FUNCTION_BLOCK FB_ComputeFromImage
VAR_INPUT
	ptrXValues	: POINTER TO ARRAY[1..GVL.NumberVisionPoints] OF REAL;
	ptrYValues	: POINTER TO ARRAY[1..GVL.NumberVisionPoints] OF REAL;
	minor		: LREAL;	// in mm
	pitch		: LREAL;	// mm per pixel
END_VAR
VAR_OUTPUT
	centerX		: LREAL;
	centerY		: LREAL;
	a			: LREAL;	// major in mm
	b			: LREAL;	// minor in mm
END_VAR
	
VAR
	fbSecond	: FB_SecondOrder;
	fbFourth	: FB_FourthOrder;
	fbEllipse	: FB_Ellipse;
	xPeak		: LREAL;
	yPeak		: LREAL;
	XMirror		: ARRAY[1..GVL.NumberEllipsePoints] OF LREAL;
	YMirror		: ARRAY[1..GVL.NumberEllipsePoints] OF LREAL;
	CenterLine	: LREAL;
	i			: INT;
END_VAR

fbSecond.FindPeak(xValues := ptrXValues, yValues := ptrYValues, xPeak := ADR(xPeak));
fbFourth.FindYatX(xValues := ptrXValues, yValues := ptrYValues, xPeak := ADR(xPeak), yPeak := ADR(yPeak));
centerLine := yPeak - (minor / pitch);

FOR i := 1 TO GVL.NumberVisionPoints DO
	XMirror[i] := REAL_TO_LREAL(ptrXValues^[i]);	
	XMirror[i + GVL.NumberVisionPoints] := REAL_TO_LREAL(ptrXValues^[i]);
	YMirror[i] := REAL_TO_LREAL(ptrYValues^[i]);
	YMirror[i + GVL.NumberVisionPoints] := REAL_TO_LREAL(ptrYValues^[i] - ABS(2*(ptrYValues^[i] - centerLine)));
END_FOR

fbEllipse.EllipseFit(xValues := xMirror, yValues := yMirror);
centerX := fbEllipse.centrex;
centerY := fbEllipse.centrey;
a := fbEllipse.major * pitch;
b := fbEllipse.minor * pitch;

END_FUNCTION_BLOCK

(* stored: Version 1.1.0.1, ProductVersion 3.1.4024.3
   POU FB_ComputeFromImage: Id {7c26fa06-d730-44cb-a3a7-f7dc14edb998}, SpecialFunc None *)
